// TIA Portal V15.1 export
// export: Created 2024-06-21T08:41:07.3517165Z, ExportSetting WithDefaults, DisplayName Totally Integrated Automation Portal, DisplayVersion V15.1 Update 5, DisplayName TIA Portal Openness, DisplayVersion V15.1 Update 5, DisplayName SINAMICS Startdrive Advanced, DisplayVersion V15.1, DisplayName G130, G150, S120, S150, SINAMICS MV, S210, DisplayVersion V15.1, DisplayName G110M, G120, G120C, G120D, G120P, DisplayVersion V15.1, DisplayName STEP 7 Professional, DisplayVersion V15.1 Update 5, DisplayName STEP 7 Safety, DisplayVersion V15.1, DisplayName WinCC Professional, DisplayVersion V15.1 Update 5, DisplayName SIMATIC Visualization Architect, DisplayVersion V15.1
FUNCTION_BLOCK "LGBFlowCodeShift"   // FB6636, FBD
TITLE = LGBFlowCodeShift
{ S7_Optimized_Access := 'TRUE' }
VERSION : 0.1
// stored: AutoNumber false, IsIECCheckEnabled false, IsRetainMemResEnabled false, MemoryReserve 100, SetENOAutomatically False, UDAEnableTagReadback false
   VAR_INPUT
      I_ArrivedToPrev1 { ExternalAccessible := 'False'; ExternalVisible := 'False'; ExternalWritable := 'False'} : Bool;   // Arrived signal to previous transfer 1
      I_FlowData1 { ExternalAccessible := 'False'; ExternalVisible := 'False'; ExternalWritable := 'False'} : Int;   // Flow data transfer 1
      I_ArrivedToPrev2 { ExternalAccessible := 'False'; ExternalVisible := 'False'; ExternalWritable := 'False'} : Bool;   // Arrived signal to previous transfer 2
      I_FlowData2 { ExternalAccessible := 'False'; ExternalVisible := 'False'; ExternalWritable := 'False'} : Int;   // Flow data transfer 2
      I_ArrivedToPrev3 { ExternalAccessible := 'False'; ExternalVisible := 'False'; ExternalWritable := 'False'} : Bool;   // Arrived signal to previous transfer 3
      I_FlowData3 { ExternalAccessible := 'False'; ExternalVisible := 'False'; ExternalWritable := 'False'} : Int;   // Flow data transfer 3
      I_ArrivedToPrev4 { ExternalAccessible := 'False'; ExternalVisible := 'False'; ExternalWritable := 'False'} : Bool;   // Arrived signal to previous transfer 4
      I_FlowData4 { ExternalAccessible := 'False'; ExternalVisible := 'False'; ExternalWritable := 'False'} : Int;   // Flow data transfer 4
      I_NextShiftDone { ExternalAccessible := 'False'; ExternalVisible := 'False'; ExternalWritable := 'False'} : Bool;   // Shift to next position is done
   END_VAR
   VAR_OUTPUT
      O_ShiftDone1 { ExternalAccessible := 'False'; ExternalVisible := 'False'; ExternalWritable := 'False'} : Bool;   // Shift done transfer 1
      O_ShiftDone2 { ExternalAccessible := 'False'; ExternalVisible := 'False'; ExternalWritable := 'False'} : Bool;   // Shift done transfer 2
      O_ShiftDone3 { ExternalAccessible := 'False'; ExternalVisible := 'False'; ExternalWritable := 'False'} : Bool;   // Shift done transfer 3
      O_ShiftDone4 { ExternalAccessible := 'False'; ExternalVisible := 'False'; ExternalWritable := 'False'} : Bool;   // Shift done transfer 4
      O_FlowData { ExternalAccessible := 'False'; ExternalVisible := 'False'; ExternalWritable := 'False'} : Int;   // Flow Data for this position
      O_AlarmABCondition { ExternalAccessible := 'False'; ExternalVisible := 'False'; ExternalWritable := 'False'} : Bool;   // Alarm AB Condition
      O_AlarmA { ExternalAccessible := 'False'; ExternalVisible := 'False'; ExternalWritable := 'False'} : Bool;   // Alarm A
      O_AlarmB { ExternalAccessible := 'False'; ExternalVisible := 'False'; ExternalWritable := 'False'} : Bool;   // Alarm B
      O_AlarmC { ExternalAccessible := 'False'; ExternalVisible := 'False'; ExternalWritable := 'False'} : Bool;   // Alarm C
      O_AlarmD { ExternalAccessible := 'False'; ExternalVisible := 'False'; ExternalWritable := 'False'} : Bool;   // Alarm D
      H_AlarmDWord { ExternalAccessible := 'False'; ExternalVisible := 'False'; ExternalWritable := 'False'} : DWord;   // HMI Animation
      H_IAnim { ExternalAccessible := 'False'; ExternalVisible := 'False'; ExternalWritable := 'False'} : DWord;   // Icon Animation
      H_IAnim2 { ExternalAccessible := 'False'; ExternalVisible := 'False'; ExternalWritable := 'False'} : DWord;   // Icon Animation
   END_VAR
   VAR_IN_OUT
      IO_Modes : "Modes";   // Modes
   END_VAR
   VAR
      AC_NoFlowData { ExternalAccessible := 'False'; ExternalVisible := 'False'; ExternalWritable := 'False'} : Bool;   // Alarm No Flow Data
      PulseArrivedToPrev1 { ExternalAccessible := 'False'; ExternalVisible := 'False'; ExternalWritable := 'False'} : Bool;   // Pulse Arrived Signal to Previous Transfer 1
      Arrived1 { ExternalAccessible := 'False'; ExternalVisible := 'False'; ExternalWritable := 'False'} : Bool;   // Arrived 1
      PulseArrivedToPrev2 { ExternalAccessible := 'False'; ExternalVisible := 'False'; ExternalWritable := 'False'} : Bool;   // Pulse Arrived Signal to Previous Transfer 2
      Arrived2 { ExternalAccessible := 'False'; ExternalVisible := 'False'; ExternalWritable := 'False'} : Bool;   // Arrived 2
      PulseArrivedToPrev3 { ExternalAccessible := 'False'; ExternalVisible := 'False'; ExternalWritable := 'False'} : Bool;   // Pulse Arrived Signal to Previous Transfer 3
      Arrived3 { ExternalAccessible := 'False'; ExternalVisible := 'False'; ExternalWritable := 'False'} : Bool;   // Arrived 3
      PulseArrivedToPrev4 { ExternalAccessible := 'False'; ExternalVisible := 'False'; ExternalWritable := 'False'} : Bool;   // Pulse Arrived Signal to Previous Transfer 4
      Arrived4 { ExternalAccessible := 'False'; ExternalVisible := 'False'; ExternalWritable := 'False'} : Bool;   // Arrived 4
   END_VAR
   VAR RETAIN
      FlowData { ExternalAccessible := 'False'; ExternalVisible := 'False'; ExternalWritable := 'False'} : Int;   // Flow Data of this position
   END_VAR
   VAR
      AlarmA { ExternalAccessible := 'False'; ExternalVisible := 'False'; ExternalWritable := 'False'} : Bool;   // Alarm A
      AlarmB { ExternalAccessible := 'False'; ExternalVisible := 'False'; ExternalWritable := 'False'} : Bool;   // Alarm B
      AlarmC { ExternalAccessible := 'False'; ExternalVisible := 'False'; ExternalWritable := 'False'} : Bool;   // Alarm C
      AlarmD { ExternalAccessible := 'False'; ExternalVisible := 'False'; ExternalWritable := 'False'} : Bool;   // Alarm D
      AlarmABCondition { ExternalAccessible := 'False'; ExternalVisible := 'False'; ExternalWritable := 'False'} : Bool;   // Alarm AB Condition
   END_VAR
   VAR_TEMP   // added for the SCL form of the ladder/FBD networks
      _w1 : Bool;
   END_VAR
BEGIN

REGION Network 1: **** 4.4 - Machine status - Calculated **** Pulse Arrived Signal 1 To previous
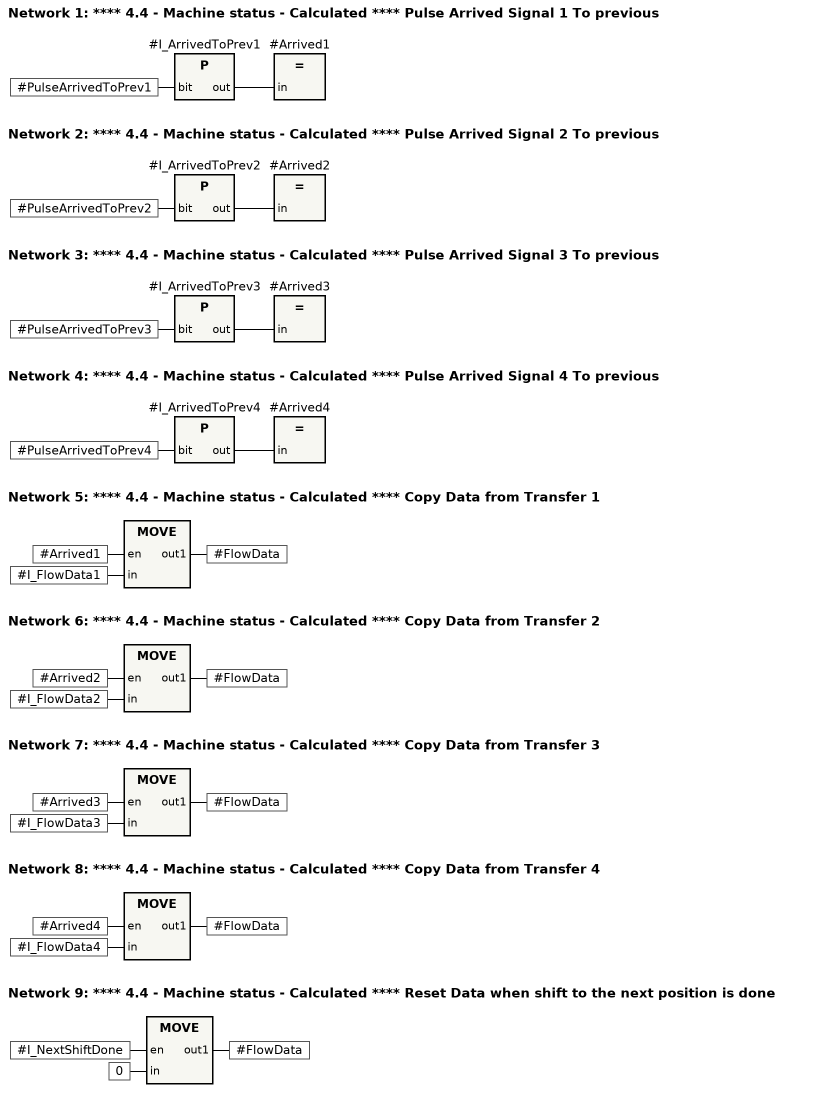
   #_w1 := #I_ArrivedToPrev1 AND NOT #PulseArrivedToPrev1;   // rising edge of #I_ArrivedToPrev1
   #PulseArrivedToPrev1 := #I_ArrivedToPrev1;
   #Arrived1 := #_w1;
END_REGION

REGION Network 2: **** 4.4 - Machine status - Calculated **** Pulse Arrived Signal 2 To previous
   #_w1 := #I_ArrivedToPrev2 AND NOT #PulseArrivedToPrev2;   // rising edge of #I_ArrivedToPrev2
   #PulseArrivedToPrev2 := #I_ArrivedToPrev2;
   #Arrived2 := #_w1;
END_REGION

REGION Network 3: **** 4.4 - Machine status - Calculated **** Pulse Arrived Signal 3 To previous
   #_w1 := #I_ArrivedToPrev3 AND NOT #PulseArrivedToPrev3;   // rising edge of #I_ArrivedToPrev3
   #PulseArrivedToPrev3 := #I_ArrivedToPrev3;
   #Arrived3 := #_w1;
END_REGION

REGION Network 4: **** 4.4 - Machine status - Calculated **** Pulse Arrived Signal 4 To previous
   #_w1 := #I_ArrivedToPrev4 AND NOT #PulseArrivedToPrev4;   // rising edge of #I_ArrivedToPrev4
   #PulseArrivedToPrev4 := #I_ArrivedToPrev4;
   #Arrived4 := #_w1;
END_REGION

REGION Network 5: **** 4.4 - Machine status - Calculated **** Copy Data from Transfer 1
   IF #Arrived1 THEN #FlowData := #I_FlowData1; END_IF;
END_REGION

REGION Network 6: **** 4.4 - Machine status - Calculated **** Copy Data from Transfer 2
   IF #Arrived2 THEN #FlowData := #I_FlowData2; END_IF;
END_REGION

REGION Network 7: **** 4.4 - Machine status - Calculated **** Copy Data from Transfer 3
   IF #Arrived3 THEN #FlowData := #I_FlowData3; END_IF;
END_REGION

REGION Network 8: **** 4.4 - Machine status - Calculated **** Copy Data from Transfer 4
   IF #Arrived4 THEN #FlowData := #I_FlowData4; END_IF;
END_REGION

REGION Network 9: **** 4.4 - Machine status - Calculated **** Reset Data when shift to the next position is done
   IF #I_NextShiftDone THEN #FlowData := 0; END_IF;
END_REGION

REGION Network 10: **** 4.6 - Machine Status - Indication **** Icon Animation
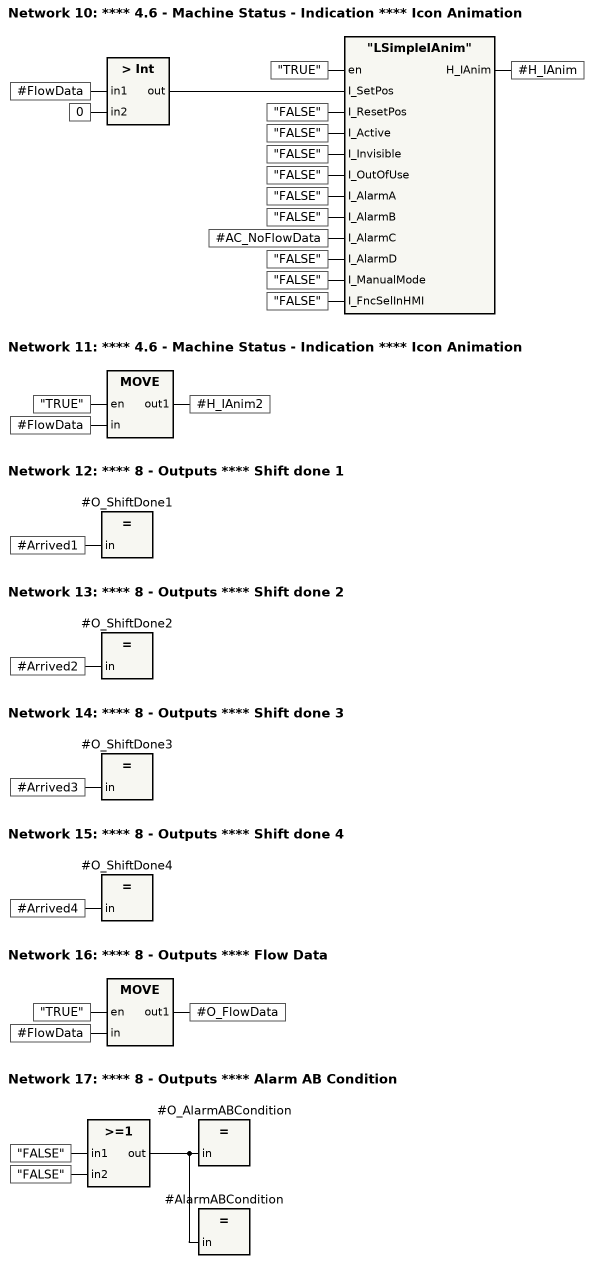
   IF "TRUE" THEN
       "LSimpleIAnim"(I_SetPos := #FlowData > 0,
                      I_ResetPos := "FALSE",
                      I_Active := "FALSE",
                      I_Invisible := "FALSE",
                      I_OutOfUse := "FALSE",
                      I_AlarmA := "FALSE",
                      I_AlarmB := "FALSE",
                      I_AlarmC := #AC_NoFlowData,
                      I_AlarmD := "FALSE",
                      I_ManualMode := "FALSE",
                      I_FncSelInHMI := "FALSE",
                      H_IAnim => #H_IAnim);
   END_IF;
END_REGION

REGION Network 11: **** 4.6 - Machine Status - Indication **** Icon Animation
   IF "TRUE" THEN #H_IAnim2 := #FlowData; END_IF;
END_REGION

REGION Network 12: **** 8 - Outputs **** Shift done 1
   #O_ShiftDone1 := #Arrived1;
END_REGION

REGION Network 13: **** 8 - Outputs **** Shift done 2
   #O_ShiftDone2 := #Arrived2;
END_REGION

REGION Network 14: **** 8 - Outputs **** Shift done 3
   #O_ShiftDone3 := #Arrived3;
END_REGION

REGION Network 15: **** 8 - Outputs **** Shift done 4
   #O_ShiftDone4 := #Arrived4;
END_REGION

REGION Network 16: **** 8 - Outputs **** Flow Data
   IF "TRUE" THEN #O_FlowData := #FlowData; END_IF;
END_REGION

REGION Network 17: **** 8 - Outputs **** Alarm AB Condition
   // Alarm AB Condition
   #O_AlarmABCondition := "FALSE" OR "FALSE";
   #AlarmABCondition := #O_AlarmABCondition;
END_REGION

REGION Network 18: **** 9 - Alarms **** Alarm no flow data
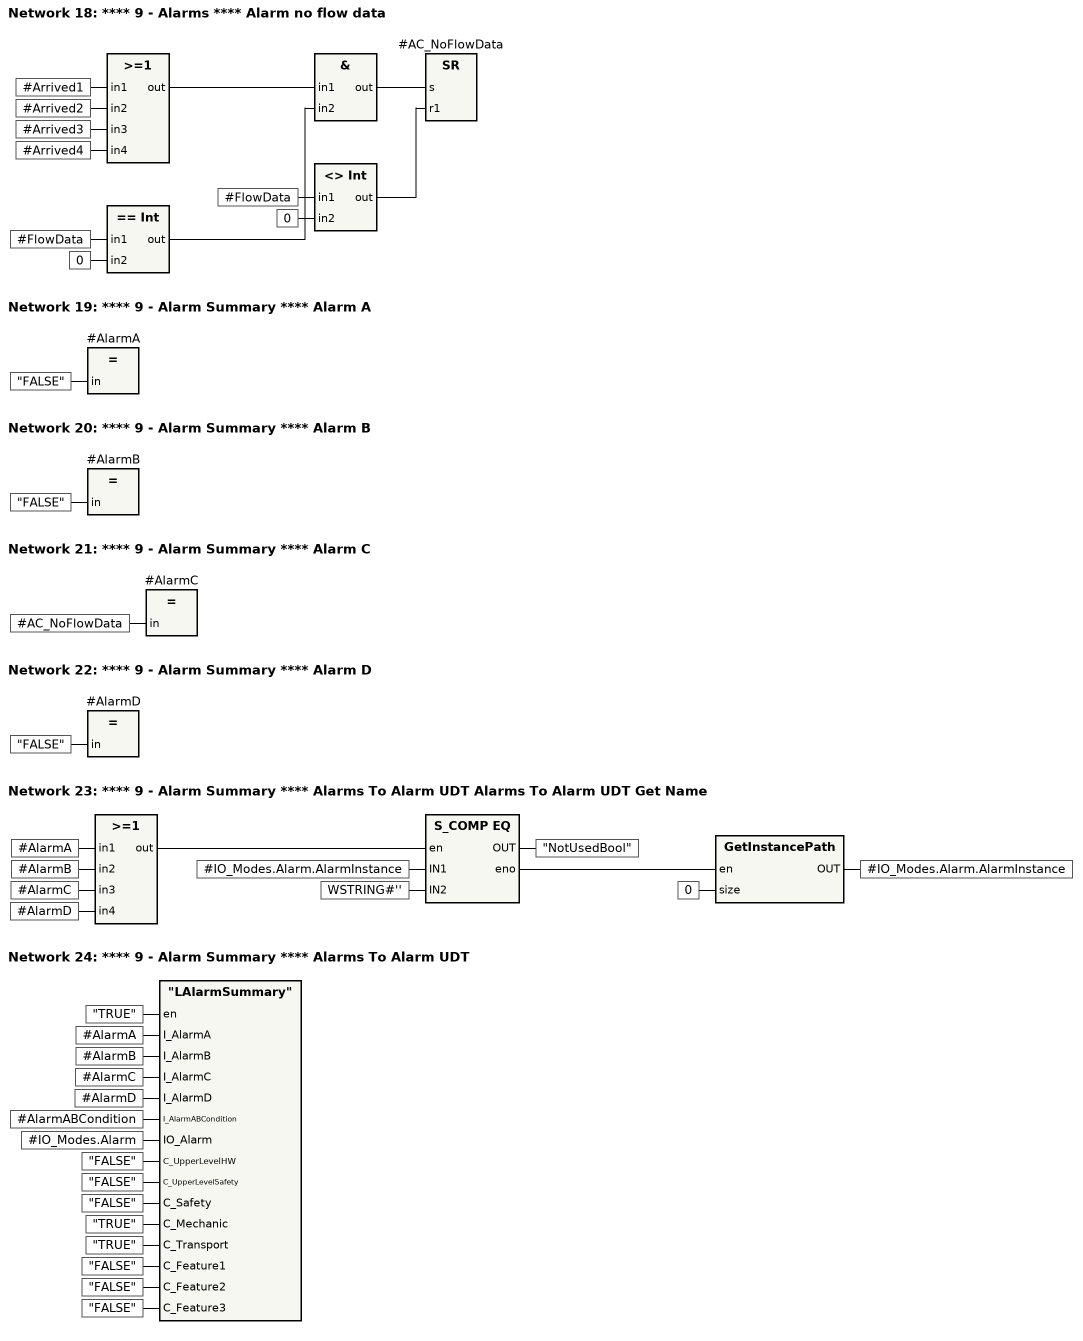
   IF (#Arrived1 OR #Arrived2 OR #Arrived3 OR #Arrived4) AND (#FlowData = 0) THEN
       #AC_NoFlowData := TRUE;   // SR flip-flop
   END_IF;
   IF #FlowData <> 0 THEN #AC_NoFlowData := FALSE; END_IF;
END_REGION

REGION Network 19: **** 9 - Alarm Summary **** Alarm A
   // Alarm A
   #AlarmA := "FALSE";
END_REGION

REGION Network 20: **** 9 - Alarm Summary **** Alarm B
   // Alarm B
   #AlarmB := "FALSE";
END_REGION

REGION Network 21: **** 9 - Alarm Summary **** Alarm C
   // Alarm C
   #AlarmC := #AC_NoFlowData;
END_REGION

REGION Network 22: **** 9 - Alarm Summary **** Alarm D
   // Alarm D
   #AlarmD := "FALSE";
END_REGION

REGION Network 23: **** 9 - Alarm Summary **** Alarms To Alarm UDT Alarms To Alarm UDT Get Name
   // Alarm D
   S_COMP(EN := #AlarmA OR #AlarmB OR #AlarmC OR #AlarmD,
          IN1 := #IO_Modes.Alarm.AlarmInstance,
          IN2 := WSTRING#'',
          OUT => "NotUsedBool",
          ENO => #_w1);
   IF #_w1 THEN GetInstancePath(size := 0, OUT => #IO_Modes.Alarm.AlarmInstance); END_IF;
END_REGION

REGION Network 24: **** 9 - Alarm Summary **** Alarms To Alarm UDT
   IF "TRUE" THEN
       "LAlarmSummary"(I_AlarmA := #AlarmA,
                       I_AlarmB := #AlarmB,
                       I_AlarmC := #AlarmC,
                       I_AlarmD := #AlarmD,
                       I_AlarmABCondition := #AlarmABCondition,
                       IO_Alarm := #IO_Modes.Alarm,
                       C_UpperLevelHW := "FALSE",
                       C_UpperLevelSafety := "FALSE",
                       C_Safety := "FALSE",
                       C_Mechanic := "TRUE",
                       C_Transport := "TRUE",
                       C_Feature1 := "FALSE",
                       C_Feature2 := "FALSE",
                       C_Feature3 := "FALSE");
   END_IF;
END_REGION

REGION Network 25: **** 9.1 - Alarm Output **** Alarm A
   // Alarm A
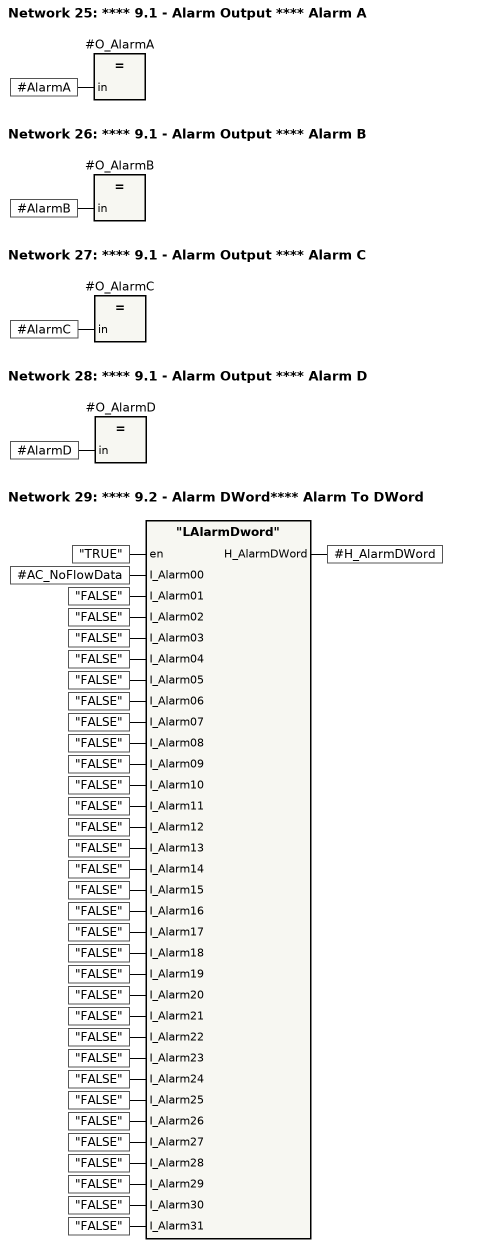
   #O_AlarmA := #AlarmA;
END_REGION

REGION Network 26: **** 9.1 - Alarm Output **** Alarm B
   // Alarm B
   #O_AlarmB := #AlarmB;
END_REGION

REGION Network 27: **** 9.1 - Alarm Output **** Alarm C
   // Alarm C
   #O_AlarmC := #AlarmC;
END_REGION

REGION Network 28: **** 9.1 - Alarm Output **** Alarm D
   // Alarm D
   #O_AlarmD := #AlarmD;
END_REGION

REGION Network 29: **** 9.2 - Alarm DWord**** Alarm To DWord
   // Alarm Word
   IF "TRUE" THEN
       "LAlarmDword"(I_Alarm00 := #AC_NoFlowData,
                     I_Alarm01 := "FALSE",
                     I_Alarm02 := "FALSE",
                     I_Alarm03 := "FALSE",
                     I_Alarm04 := "FALSE",
                     I_Alarm05 := "FALSE",
                     I_Alarm06 := "FALSE",
                     I_Alarm07 := "FALSE",
                     I_Alarm08 := "FALSE",
                     I_Alarm09 := "FALSE",
                     I_Alarm10 := "FALSE",
                     I_Alarm11 := "FALSE",
                     I_Alarm12 := "FALSE",
                     I_Alarm13 := "FALSE",
                     I_Alarm14 := "FALSE",
                     I_Alarm15 := "FALSE",
                     I_Alarm16 := "FALSE",
                     I_Alarm17 := "FALSE",
                     I_Alarm18 := "FALSE",
                     I_Alarm19 := "FALSE",
                     I_Alarm20 := "FALSE",
                     I_Alarm21 := "FALSE",
                     I_Alarm22 := "FALSE",
                     I_Alarm23 := "FALSE",
                     I_Alarm24 := "FALSE",
                     I_Alarm25 := "FALSE",
                     I_Alarm26 := "FALSE",
                     I_Alarm27 := "FALSE",
                     I_Alarm28 := "FALSE",
                     I_Alarm29 := "FALSE",
                     I_Alarm30 := "FALSE",
                     I_Alarm31 := "FALSE",
                     H_AlarmDWord => #H_AlarmDWord);
   END_IF;
END_REGION
END_FUNCTION_BLOCK
